// TIA Portal V20 export
DATA_BLOCK "SP202"   // DB313
// stored: MemoryReserve 100
   VAR
      "MAIN OP AUTO INITIATE PBL LAMP ON (GREEN)" : Bool;
      "MAIN OP STOP PBL LAMP ON (RED)" : Bool;
      RESERVE : Bool;
      "MAIN OP ENABLE PBL LAMP ON (WHITE)" : Bool;
      "MAIN OP SAFETY RESET PBL LAMP ON (BLUE)" : Bool;
      SPARE : Bool;
      SPARE_1 : Bool;
      SPARE_2 : Bool;
      "TOWER LAMP 1 ON (RED)" : Bool;
      "TOWER LAMP 2 ON (AMBER)" : Bool;
      "TOWER LAMP 3 ON (GREEN)" : Bool;
      "TOWER LAMP 4 ON (WHITE)" : Bool;
      "TOWER LAMP 5 ON (BLUE)" : Bool;
      "TOWER LAMP BUZZER ON" : Bool;
      SPARE_3 : Bool;
      SPARE_4 : Bool;
   END_VAR
BEGIN
END_DATA_BLOCK
